// Mitsubishi GX Works2 project: BookEX6_37 Buffer   PLC: Q13UDV

// global labels: Global
VAR_GLOBAL
  bVar0 AT M5000 : BOOL;
  abArray0 AT M5010 : ARRAY [0..49] OF BOOL;
  sStr0 AT D5000 : STRING[199];
  sStr1 AT D5100 : STRING[199];
  sStr2 AT D5200 : STRING[199];
  sStr3 AT D5300 : STRING[199];
  sStr4 AT D5400 : STRING[199];
  sStr5 AT D5500 : STRING[199];
  sStr6 AT D5600 : STRING[199];
  sStr7 AT D5700 : STRING[199];
  sStr8 AT D5800 : STRING[199];
  sStr9 AT D5900 : STRING[199];
  iVar0 AT D4500 : INT;
  iVar1 AT D4501 : INT;
  iVar2 AT D4502 : INT;
  iVar3 AT D4503 : INT;
  iVar4 AT D4504 : INT;
  iVar5 AT D4505 : INT;
  iVar6 AT D4506 : INT;
  iVar7 AT D4507 : INT;
  iVar8 AT D4508 : INT;
  iVar9 AT D4509 : INT;
  dVar0 AT D4510 : DINT;
  dVar1 AT D4512 : DINT;
  dVar2 AT D4514 : DINT;
  dVar3 AT D4516 : DINT;
  dVar4 AT D4518 : DINT;
  dVar5 AT D4520 : DINT;
  dVar6 AT D4522 : DINT;
  dVar7 AT D4524 : DINT;
  dVar8 AT D4526 : DINT;
  dVar9 AT D4528 : DINT;
  wVar0 AT D4530 : WORD;
  wVar1 AT D4531 : WORD;
  wVar2 AT D4532 : WORD;
  wVar3 AT D4533 : WORD;
  wVar4 AT D4534 : WORD;
  wVar5 AT D4535 : WORD;
  wVar6 AT D4536 : WORD;
  wVar7 AT D4537 : WORD;
  wVar8 AT D4538 : WORD;
  wVar9 AT D4539 : WORD;
  dwVar0 AT D4540 : DWORD;
  dwVar1 AT D4542 : DWORD;
  dwVar2 AT D4544 : DWORD;
  dwVar3 AT D4546 : DWORD;
  dwVar4 AT D4548 : DWORD;
  dwVar5 AT D4550 : DWORD;
  dwVar6 AT D4552 : DWORD;
  dwVar7 AT D4554 : DWORD;
  dwVar8 AT D4556 : DWORD;
  dwVar9 AT D4558 : DWORD;
  fsVar0 AT D4560 : REAL;
  fsVar1 AT D4562 : REAL;
  fsVar2 AT D4564 : REAL;
  fsVar3 AT D4566 : REAL;
  fsVar4 AT D4568 : REAL;
  fsVar5 AT D4570 : REAL;
  fsVar6 AT D4572 : REAL;
  fsVar7 AT D4574 : REAL;
  fsVar8 AT D4576 : REAL;
  fsVar9 AT D4578 : REAL;
  fdVar0 AT D4580 : LREAL;
  tTime0 AT D4620 : TIME;
  tTime1 AT D4622 : TIME;
  tTime2 AT D4624 : TIME;
  tTime3 AT D4626 : TIME;
  tTime4 AT D4628 : TIME;
  tTime5 AT D4630 : TIME;
  tTime6 AT D4632 : TIME;
  tTime7 AT D4634 : TIME;
  tTime8 AT D4636 : TIME;
  tTime9 AT D4638 : TIME;
  tTime10 AT D4640 : TIME;
  bVar1 AT M5001 : BOOL;
  bVar2 AT M5002 : BOOL;
  bVar3 AT M5003 : BOOL;
  bVar4 AT M5004 : BOOL;
  bVar5 AT M5005 : BOOL;
  bVar6 AT M5006 : BOOL;
  bVar7 AT M5007 : BOOL;
  bVar8 AT M5008 : BOOL;
  bVar9 AT M5009 : BOOL;
  abArray1 AT M5060 : ARRAY [0..49] OF BOOL;
  abArray2 AT M5110 : ARRAY [0..49] OF BOOL;
  abArray3 AT M5160 : ARRAY [0..49] OF BOOL;
  abArray4 AT M5210 : ARRAY [0..49] OF BOOL;
  abArray5 AT M5260 : ARRAY [0..49] OF BOOL;
  abArray6 AT M5310 : ARRAY [0..49] OF BOOL;
  abArray7 AT M5360 : ARRAY [0..49] OF BOOL;
  abArray8 AT M5410 : ARRAY [0..49] OF BOOL;
  abArray9 AT M5460 : ARRAY [0..49] OF BOOL;
  fdVar1 AT D4584 : LREAL;
  fdVar2 AT D4588 : LREAL;
  fdVar3 AT D4592 : LREAL;
  fdVar4 AT D4596 : LREAL;
  fdVar5 AT D4600 : LREAL;
  fdVar6 AT D4604 : LREAL;
  fdVar7 AT D4608 : LREAL;
  fdVar8 AT D4612 : LREAL;
  fdVar9 AT D4616 : LREAL;
  afsPen0 AT D2000 : ARRAY [0..499] OF REAL;
  afsPen1 AT D3000 : ARRAY [0..499] OF REAL;
END_VAR
// user libraries (not included): HMI

FUNCTION_BLOCK cntEqu
VAR_INPUT
  b_EN : BOOL;
END_VAR
VAR
  bError : BOOL;
  bReady : BOOL;
  bRes : BOOL;
END_VAR
VAR_INPUT
  i_Start_IO : INT;
END_VAR
VAR_OUTPUT
  b_ENO : BOOL;
END_VAR
VAR_INPUT
  b_Set : BOOL;
  d_SetVal : DINT;
  b_Reset : BOOL;
END_VAR
VAR_OUTPUT
  b_Large : BOOL;
  b_Equ : BOOL;
  b_Small : BOOL;
END_VAR
;
b_ENO := b_EN;
IF NOT b_EN THEN
	RETURN;
END_IF;
(* Status *)
Z0 := i_Start_IO * 16;
bError := X0FZ0;
bReady := X00Z0;
	
IF LDP(TRUE, b_Set) AND NOT bError AND bReady THEN
	bRes := DTO(TRUE , d_SetVal, i_Start_IO , 4 , 1 );	
	DELTA(TRUE, DY00Z0);	(* Reset *)
	Y02Z0 := TRUE;						(* 허가*) 
END_IF;
	
IF bReady THEN
	IF Y02Z0 AND X02Z0 AND NOT Y0Z0 THEN
		b_Equ := TRUE;
	END_IF;
	IF X2Z0 AND b_Reset THEN
		Y0Z0 := TRUE;
	END_IF;
	IF NOT X2Z0 AND Y0Z0 THEN
		Y0Z0 := FALSE;
	END_IF;
END_IF;
b_Large := X1Z0;
b_Equ := X2Z0;
b_Small := X3Z0;
END_FUNCTION_BLOCK

FUNCTION_BLOCK cntFunction
VAR_INPUT
  b_EN : BOOL;
END_VAR
VAR
  bError : BOOL;
  bReady : BOOL;
  bRes : BOOL;
END_VAR
VAR_INPUT
  i_Start_IO : INT;
END_VAR
VAR_OUTPUT
  b_ENO : BOOL;
END_VAR
VAR_INPUT
  b_Set : BOOL;
  i_Func : INT;
END_VAR
VAR_OUTPUT
  b_Run : BOOL;
  d_Latch : DINT;
  d_Sample : DINT;
  d_PeriodP : DINT;
  d_PeriodC : DINT;
END_VAR
VAR_INPUT
  i_SampTime : INT;
  b_Read : BOOL;
END_VAR
;
b_ENO := b_EN;
IF NOT b_EN THEN
	RETURN;
END_IF;
(* Status *)
Z0 := i_Start_IO * 16;
bError := X0FZ0;
bReady := X00Z0;

IF LDP(TRUE, b_Set) AND NOT bError AND bReady THEN
	CASE i_Func OF
		0 : (* No Count *)
			bRes := TOP(TRUE, 0, i_Start_IO , 9 , 1 );	
			Y6Z0 := TRUE;
		1 : (* Latch *)
			bRes := TOP(TRUE, 1, i_Start_IO , 9 , 1 );	
			Y6Z0 := TRUE;
(* PLS(TRUE, Y6Z0); *)
		2 : (* Sampling *)
			bRes := TOP(TRUE, i_SampTime, i_Start_IO , 10 , 1 );	
			bRes := TOP(TRUE, 2, i_Start_IO , 9 , 1 );	
			Y6Z0 := TRUE;
		3 : (* Period *)
			bRes := TOP(TRUE, i_SampTime, i_Start_IO , 10 , 1 );	
			bRes := TOP(TRUE, 3, i_Start_IO , 9 , 1 );	
			Y6Z0 := TRUE;
	ELSE
			Y6Z0 := FALSE;
	END_CASE;
END_IF;
	
(* Data Read *)
IF b_Read AND NOT bError AND bReady THEN
	CASE i_Func OF
		1 : (* Latch *)
			bRes := DFRO(TRUE , i_Start_IO , 12 , 1 , d_Latch);
		2 : (* Sampling *)
			bRes := DFRO(TRUE , i_Start_IO , 14 , 1 , d_Sample);
		3 : (* Period *)
			bRes := DFRO(TRUE , i_Start_IO , 16 , 1 , d_PeriodP);
			bRes := DFRO(TRUE , i_Start_IO , 18 , 1 , d_PeriodC);
	END_CASE;
END_IF;
b_Run := Y6Z0;
END_FUNCTION_BLOCK

FUNCTION_BLOCK cntRead
VAR_INPUT
  b_EN : BOOL;
END_VAR
VAR_IN_OUT
  b_InitDone : BOOL;
END_VAR
VAR_OUTPUT
  b_Error : BOOL;
  b_Ready : BOOL;
END_VAR
VAR
  bRes : BOOL;
  SeqInit : INT;
  Buffer1 : DINT;
END_VAR
VAR_INPUT
  i_Start_IO : INT;
END_VAR
VAR_OUTPUT
  b_ENO : BOOL;
  d_Cnt1 : DINT;
  d_Cnt2 : DINT;
END_VAR
VAR
  Buffer2 : DINT;
END_VAR
VAR_INPUT
  b_Reset1 : BOOL;
  b_Reset2 : BOOL;
END_VAR
;
b_ENO := b_EN;
IF NOT b_EN THEN
	RETURN;
END_IF;

Z0 := i_Start_IO * 16;
b_Error := X0FZ0;
b_Ready := X00Z0;

CASE SeqInit OF
	0 : 
		IF NOT b_InitDone AND NOT b_Error  THEN
			SeqInit := 1;
		END_IF;
	1 : 
		IF b_Ready THEN
			bRes := DTO(TRUE , 0, i_Start_IO , 0 , 1 );
			bRes := DTO(TRUE , 0, i_Start_IO , 32 , 1 );
			Y04Z0 := TRUE;
			Y0CZ0 := TRUE;
			SeqInit := 2;
		END_IF;
	2 : 
		b_InitDone := TRUE;
		SeqInit := 100;
END_CASE;
Y01Z0 := b_Reset1;
Y09Z0 := b_Reset2;
	
IF b_InitDone AND b_Ready THEN
	bRes := DFRO(TRUE , i_Start_IO , 2 , 1 , Buffer1);
	bRes := DFRO(TRUE , i_Start_IO , 34 , 1 , Buffer2);
	d_Cnt1 := Buffer1; 
	d_Cnt2 := Buffer2; 
END_IF;
END_FUNCTION_BLOCK

FUNCTION_BLOCK cntStop
VAR_INPUT
  b_EN : BOOL;
  i_Start_IO : INT;
END_VAR
VAR_OUTPUT
  b_ENO : BOOL;
END_VAR
VAR_INPUT
  b_Run1 : BOOL;
  b_Run2 : BOOL;
END_VAR
VAR
  bError : BOOL;
  bReady : BOOL;
END_VAR
;
b_ENO := b_EN;
IF NOT b_EN THEN
	RETURN;
END_IF;

Z0 := i_Start_IO * 16;
bError := X0FZ0;
bReady := X00Z0;

IF NOT bError  AND bReady THEN
	Y04Z0 := b_Run1;
	Y0CZ0 := b_Run2;
END_IF;
END_FUNCTION_BLOCK

PROGRAM ExBARCODE
(* structured ladder/FBD written out as ST: instructions are called as NAME(EN, inputs, outputs); _pN, _eN, _tN stand for wires *)
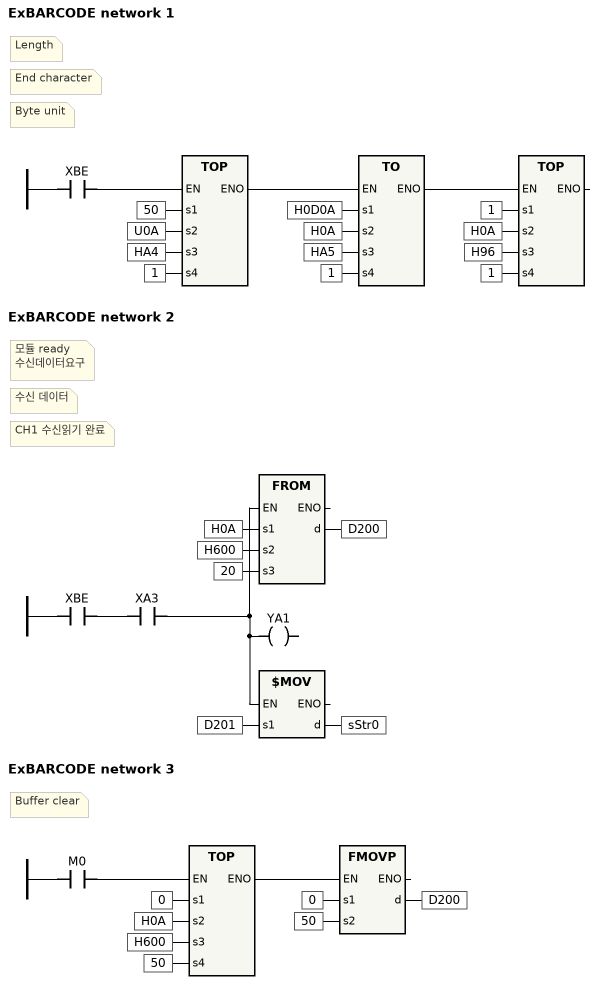
(* network 1 *)
(* Length *)
(* End character *)
(* Byte unit *)
_e1 := TOP(XBE, 50, U0A, HA4, 1);
_e2 := TO(_e1, H0D0A, H0A, HA5, 1);
TOP(_e2, 1, H0A, H96, 1);
(* network 2 *)
(* 모듈 ready / 수신데이터요구 *)
(* 수신 데이터 *)
(* CH1 수신읽기 완료 *)
_p1 := XBE AND XA3;
FROM(_p1, H0A, H600, 20, D200);
YA1 := _p1;
$MOV(_p1, D201, sStr0);
(* network 3 *)
(* Buffer clear *)
_e1 := TOP(M0, 0, H0A, H600, 50);
FMOVP(_e1, 0, 50, D200);
END_PROGRAM

PROGRAM ExFROM
(* structured ladder/FBD written out as ST: instructions are called as NAME(EN, inputs, outputs); _pN, _eN, _tN stand for wires *)
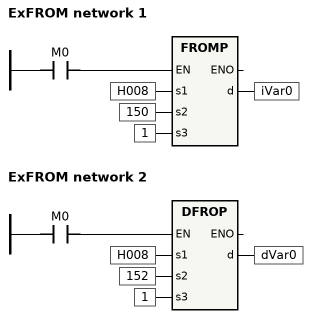
(* network 1 *)
FROMP(M0, H008, 150, 1, iVar0);
(* network 2 *)
DFROP(M0, H008, 152, 1, dVar0);
END_PROGRAM

PROGRAM ExQD62D
VAR
  cntRead_1 : cntRead;
  bInit : BOOL;
  bError : BOOL;
  bReady : BOOL;
  CH1counter : DINT;
  CH2counter : DINT;
  cntStop_1 : cntStop;
  cntEqu_1 : cntEqu;
  bEQU : BOOL;
  bLarge : BOOL;
  bSmall : BOOL;
  cntFunction_1 : cntFunction;
  bRun : BOOL;
  dLatch : DINT;
  dSample : DINT;
  dPeriodC : DINT;
  dPeriodP : DINT;
END_VAR
(* structured ladder/FBD written out as ST: instructions are called as NAME(EN, inputs, outputs); _pN, _eN, _tN stand for wires *)
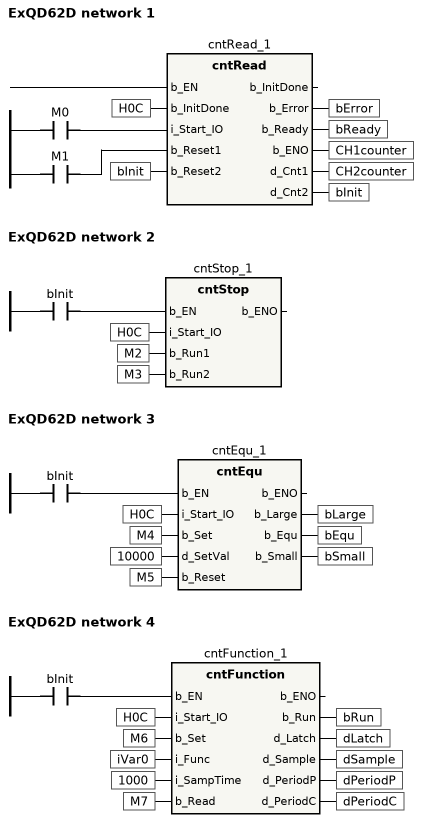
(* network 1 *)
cntRead_1(b_EN := TRUE, b_InitDone := H0C, i_Start_IO := M0, b_Reset1 := M1, b_Reset2 := bInit, b_Error => bError, b_Ready => bReady, b_ENO => CH1counter, d_Cnt1 => CH2counter, d_Cnt2 => bInit);
(* network 2 *)
cntStop_1(b_EN := bInit, i_Start_IO := H0C, b_Run1 := M2, b_Run2 := M3);
(* network 3 *)
cntEqu_1(b_EN := bInit, i_Start_IO := H0C, b_Set := M4, d_SetVal := 10000, b_Reset := M5, b_Large => bLarge, b_Equ => bEqu, b_Small => bSmall);
(* network 4 *)
cntFunction_1(b_EN := bInit, i_Start_IO := H0C, b_Set := M6, i_Func := iVar0, i_SampTime := 1000, b_Read := M7, b_Run => bRun, d_Latch => dLatch, d_Sample => dSample, d_PeriodP => dPeriodP, d_PeriodC => dPeriodC);
END_PROGRAM

PROGRAM ExTO
(* structured ladder/FBD written out as ST: instructions are called as NAME(EN, inputs, outputs); _pN, _eN, _tN stand for wires *)
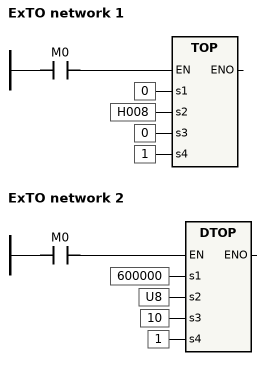
(* network 1 *)
TOP(M0, 0, H008, 0, 1);
(* network 2 *)
DTOP(M0, 600000, U8, 10, 1);
END_PROGRAM

PROGRAM ExBook
VAR
  bMreg : BOOL;
  Mov4INT_1 : Mov4INT;
  Mov8INT_1 : Mov8INT;
END_VAR
(* structured ladder/FBD written out as ST: instructions are called as NAME(EN, inputs, outputs); _pN, _eN, _tN stand for wires *)
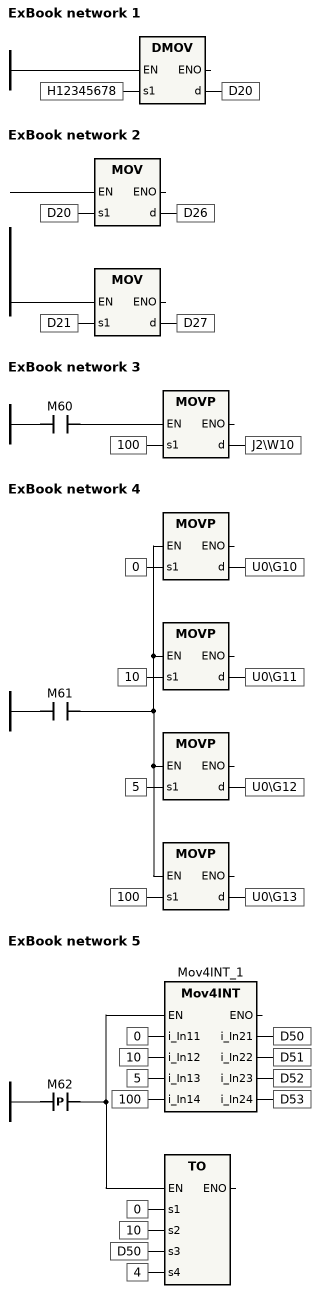
(* network 1 *)
DMOV(TRUE, H12345678, D20);
(* network 2 *)
MOV(TRUE, D20, D26);
MOV(TRUE, D21, D27);
(* network 3 *)
MOVP(M60, 100, J2\W10);
(* network 4 *)
MOVP(M61, 0, U0\G10);
MOVP(M61, 10, U0\G11);
MOVP(M61, 5, U0\G12);
MOVP(M61, 100, U0\G13);
(* network 5 *)
_p1 := LDP(TRUE, M62);
Mov4INT_1(EN := _p1, i_In11 := 0, i_In12 := 10, i_In13 := 5, i_In14 := 100, i_In21 => D50, i_In22 => D51, i_In23 => D52, i_In24 => D53);
TO(_p1, 0, 10, D50, 4);
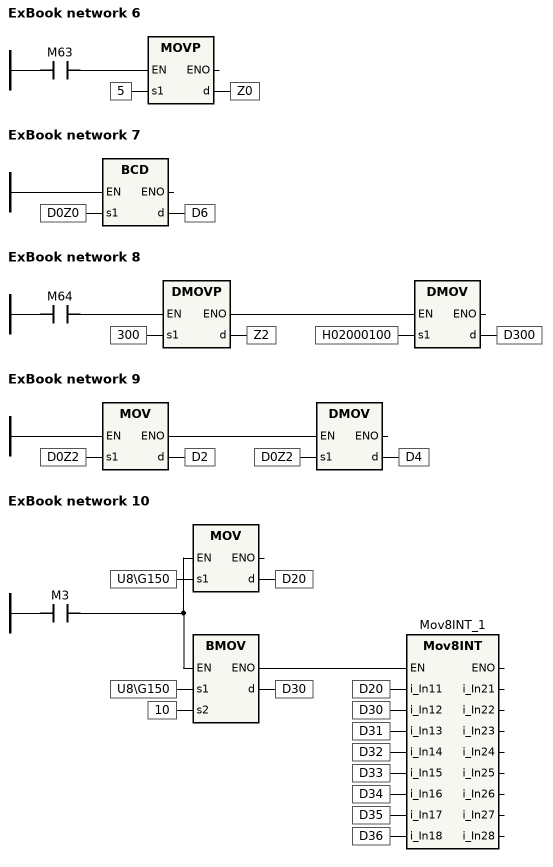
(* network 6 *)
MOVP(M63, 5, Z0);
(* network 7 *)
BCD(TRUE, D0Z0, D6);
(* network 8 *)
_e1 := DMOVP(M64, 300, Z2);
DMOV(_e1, H02000100, D300);
(* network 9 *)
_e1 := MOV(TRUE, D0Z2, D2);
DMOV(_e1, D0Z2, D4);
(* network 10 *)
MOV(M3, U8\G150, D20);
_e1 := BMOV(M3, U8\G150, 10, D30);
Mov8INT_1(EN := _e1, i_In11 := D20, i_In12 := D30, i_In13 := D31, i_In14 := D32, i_In15 := D33, i_In16 := D34, i_In17 := D35, i_In18 := D36);
END_PROGRAM
